(* PLC project Generated.project, CODESYS CODESYS V3.5 SP19 Patch 1 *)
(* stored: creationDateTime 2026-09-01T00:57:57.753728, modificationDateTime 2026-09-01T00:57:57.753728 *)

(* ═══════════════════════════════════════════════════════════════ 🪨 ST_CycleDiveSearchHMI — Échange IHM cycle plongée (DiveSearch) ═══════════════════════════════════════════════════════════════ *)
TYPE ST_CycleDiveSearchHMI : STRUCT
  Cmd : ST_CycleDiveSearchCmd;
  State : ST_CycleDiveSearchState;
  Cfg : ST_CycleDiveSearchCfg;
END_STRUCT;
END_TYPE

(* ═══════════════════════════════════════════════════════════════ ⚙️ ST_CycleDiveSearchCfg — Réglages persistants cycle plongée (DiveSearch) 📄 Doc : DOC/AF/AF_Partie-04_Mode_SemiAuto_Sequenceur_v2.3.md §3ter ═══════════════════════════════════════════════════════════════ *)
TYPE ST_CycleDiveSearchCfg : STRUCT
  DiveStartMin_M : REAL := 1;  (* Position mini M1/M2 avant plongée *)
  ImmersionUpper_M : REAL := 0.5;  (* Borne haute fenêtre front immersion *)
  ImmersionLower_M : REAL := -0.5;  (* Borne basse fenêtre front immersion *)
  Initialized : BOOL := FALSE;  (* 🚦 flag restauration boot *)
END_STRUCT;
END_TYPE

(* ═══════════════════════════════════════════════════════════════ 🎮 ST_CycleDiveSearchCmd — Sélections IHM cycle plongée (DiveSearch) ═══════════════════════════════════════════════════════════════ *)
TYPE ST_CycleDiveSearchCmd : STRUCT
  TglEnableDiveSearch : BOOL := FALSE;  (* Assistance plongée active *)
  TglBypassDiveSearchSequence : BOOL := FALSE;  (* Bypass séquence DiveSearch *)
  TglBucketAtBottomConfirmed : BOOL := FALSE;  (* Attestation manuelle fond *)
END_STRUCT;
END_TYPE

(* ═══════════════════════════════════════════════════════════════ 🚦 ST_CycleDiveSearchState — États publics cycle plongée (DiveSearch) ═══════════════════════════════════════════════════════════════ *)
TYPE ST_CycleDiveSearchState : STRUCT
  DiveReady : BOOL;
  DiveBusy : BOOL;
  DiveDone : BOOL;
  DiveError : BOOL;
  DiveErrorId : WORD;
  DiveState : E_DiveSearchState;
  DiveStepAtFault : E_DiveSearchState;
  BottomTouchConfirmed : BOOL;
  BypassDiveActive : BOOL;  (* TglBypassDiveSearchSequence armé (descente couplée en cours) *)
  BypassKoboldBottomTouched : BOOL;  (* Fond confirmé par le bypass (front montant Kobold en descente) *)
  OperatorActionId : WORD;  (* Une seule consigne conduite, arbitré en PRG_03 *)
  OperatorAction : STRING(120);  (* Texte de secours ; IHM peut mapper l'identifiant *)
END_STRUCT;
END_TYPE
